RoboDK station: Entorno1_4clases.rdk

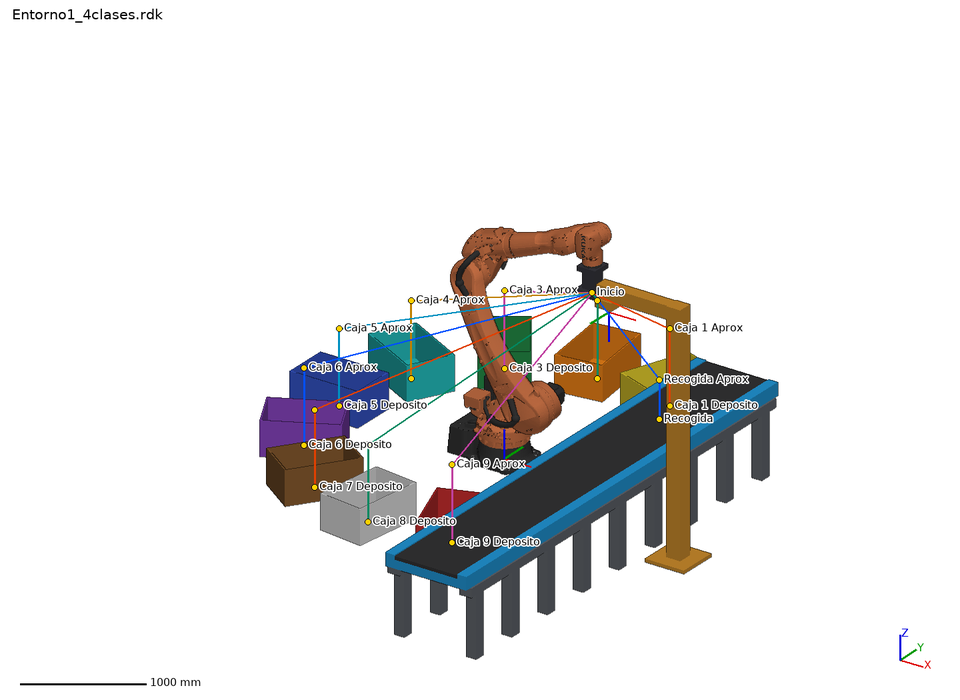
[picture v0: the station drawn from its stored meshes, robots at their saved joint values, targets as dots, program paths as lines]
Station Entorno1 (saved by RoboDK 5.9.0). Poses are relative to the parent item; angles as X-Y-Z fixed-axis rotations.
Station parameters (name, value as stored): BandaEstado, OFF, PRUEBA_LLAMADA, fin, TIPO_B0, 0, TIPO_B1, 1, TIPO_B2, 0, TIPO_B3, 0, TIPO_VALIDO, 0, HOJA_EN_CAMARA, 0, ORDEN_RECIBIDA, 0, ROBOT_OCUPADO, 0, CAJA_DESTINO, 2, ULTIMO_CODIGO, 2, VENTOSA, 0, CONTROL, RUN, IMAGEN_HOJA, C:/Users/edgar/OneDrive/Escritorio/RoboDK\camara_hoja_actual.png, HOJA_ID, 20260911_153832767_iOS
  - frame KUKA IONTEC ultra KR 120 R2700 Base at (0, 0, 0) mm
    - robot KUKA IONTEC ultra KR 120 R2700: 6 axes
        modified DH rows (alpha deg, a mm, theta deg, d mm): 0, 0, 0, 575; -90, 330, 0, 0; 0, 1180, -90, 0; -90, 170, 0, 1180; 90, 0, 0, 0; -90, 0, 180, 230
        joint limits [-185, -140, -95, -180, -125, -350] to [185, 60, 171, 180, 125, 350]; home [0, -90, 90, 0, 0, 0]; saved at [0, -117, 97.5, 0, 109.5, 0]
      - tool Ventosa, TCP at (0, 0, 250) mm, size 200 x 200 x 250 mm
  - object Banda at (0, 0, 0) mm, size 606 x 4306 x 30 mm
  - object Banda Bastidor at (0, 0, 0) mm, size 786 x 4306 x 120 mm
  - object Soporte Banda at (0, 0, 0) mm, size 816 x 4206 x 656.5 mm
  - object Estructura Camara at (0, 0, 0) mm, size 940 x 380 x 2242.1 mm
    - frame Camara Ref at (1500, -700, 1992.06) mm, rotated rx 180 ry 0 rz 0 deg
  - camera Camara Banda
  - object Caja 1 at (547.23, 1503.51, 0) mm, rotated rx 0 ry 0 rz 70 deg, size 660 x 430 x 320 mm
  - object Caja 2 at (-208.84, 1586.31, 0) mm, rotated rx 0 ry 0 rz 97.5 deg, size 660 x 430 x 320 mm
    - object Hoja 5 - connecticut capa at (-277.68, 0, 15) mm, rotated rx 0 ry 0 rz -90 deg, size 264.4 x 555.4 x 0.3 mm, geometry from 20260911_152855641_iOS.obj
    - object Hoja 6 - connecticut capa at (-259.95, 0, 15) mm, rotated rx 0 ry 0 rz -90 deg, size 208.9 x 519.9 x 0.3 mm, geometry from 20260911_153551286_iOS.obj
    - object Hoja 10 - connecticut capa at (-280.67, 0, 15) mm, rotated rx 0 ry 0 rz -90 deg, size 309.3 x 561.3 x 0.3 mm, geometry from 20260911_152611302_iOS.obj
    - object Hoja 14 - connecticut capa at (-290.65, 0, 15) mm, rotated rx 0 ry 0 rz -90 deg, size 317.9 x 581.3 x 0.3 mm, geometry from 20260911_152947681_iOS.obj
    - object Hoja 15 - connecticut capa at (-210.73, 0, 15) mm, rotated rx 0 ry 0 rz -90 deg, size 202 x 421.5 x 0.3 mm, geometry from 20260911_152212891_iOS.obj
    - object Hoja 16 - connecticut capa at (-248.11, 0, 15) mm, rotated rx 0 ry 0 rz -90 deg, size 209.5 x 496.2 x 0.3 mm, geometry from 20260911_154449975_iOS.obj
    - object Hoja 17 - connecticut capa at (-297.04, 0, 15) mm, rotated rx 0 ry 0 rz -90 deg, size 321 x 594.1 x 0.3 mm, geometry from 20260911_152508518_iOS.obj
    - object Hoja 18 - connecticut capa at (-263.19, 0, 15) mm, rotated rx 0 ry 0 rz -90 deg, size 219.7 x 526.4 x 0.3 mm, geometry from 20260911_152643389_iOS.obj
    - object Hoja 20 - connecticut capa at (-262.17, 0, 15) mm, rotated rx 0 ry 0 rz -90 deg, size 238.9 x 524.3 x 0.3 mm, geometry from 20260911_153832767_iOS.obj
  - object Caja 3 at (-917.72, 1310.64, 0) mm, rotated rx 0 ry 0 rz 125 deg, size 660 x 430 x 320 mm
    - object Hoja 1 - connecticut xl_izq at (-252.38, 0, 15) mm, rotated rx 0 ry 0 rz -90 deg, size 223.1 x 504.8 x 0.3 mm, geometry from 20260911_160812762_iOS.obj
    - object Hoja 7 - connecticut xl_izq at (-285.08, 0, 15) mm, rotated rx 0 ry 0 rz -90 deg, size 179.8 x 570.2 x 0.3 mm, geometry from 20260911_160352812_iOS.obj
    - object Hoja 13 - connecticut xl_izq at (-242.13, 0, 15) mm, rotated rx 0 ry 0 rz -90 deg, size 175.8 x 484.3 x 0.3 mm, geometry from 20260911_155539515_iOS.obj
  - object Caja 4 at (-1419.22, 738.8, 0) mm, rotated rx 0 ry 0 rz 152.5 deg, size 660 x 430 x 320 mm
    - object Hoja 9 - connecticut xr_der at (-263.12, 0, 15) mm, rotated rx 0 ry 0 rz -90 deg, size 209.2 x 526.2 x 0.3 mm, geometry from 20260911_161335259_iOS.obj
  - object Caja 5 at (-1600, 0, 0) mm, rotated rx 0 ry 0 rz 180 deg, size 660 x 430 x 320 mm
  - object Caja 6 at (-1419.22, -738.8, 0) mm, rotated rx 0 ry 0 rz -152.5 deg, size 660 x 430 x 320 mm
  - object Caja 7 at (-917.72, -1310.64, 0) mm, rotated rx 0 ry 0 rz -125 deg, size 660 x 430 x 320 mm
  - object Caja 8 at (-208.84, -1586.31, 0) mm, rotated rx 0 ry 0 rz -97.5 deg, size 660 x 430 x 320 mm
  - object Caja 9 at (547.23, -1503.51, 0) mm, rotated rx 0 ry 0 rz -70 deg, size 660 x 430 x 320 mm
    - object Hoja 2 - connecticut xl_izq at (-271.25, 0, 15) mm, rotated rx 0 ry 0 rz -90 deg, size 221.9 x 542.5 x 0.3 mm, geometry from 20260911_160413627_iOS.obj
    - object Hoja 3 - connecticut xr_der at (-283.84, 0, 15) mm, rotated rx 0 ry 0 rz -90 deg, size 206.1 x 567.7 x 0.3 mm, geometry from 20260911_161114446_iOS.obj
    - object Hoja 4 - connecticut xr_der at (-251.64, 0, 15) mm, rotated rx 0 ry 0 rz -90 deg, size 209.9 x 503.3 x 0.3 mm, geometry from 20260911_161042953_iOS.obj
    - object Hoja 8 - connecticut xl_izq at (-249.2, 0, 15) mm, rotated rx 0 ry 0 rz -90 deg, size 190.4 x 498.4 x 0.3 mm, geometry from 20260911_160151563_iOS.obj
    - object Hoja 11 - connecticut xr_der at (-278.06, 0, 15) mm, rotated rx 0 ry 0 rz -90 deg, size 229.2 x 556.1 x 0.3 mm, geometry from 20260911_161421883_iOS.obj
    - object Hoja 12 - connecticut capa at (-311.99, 0, 15) mm, rotated rx 0 ry 0 rz -90 deg, size 292.7 x 624 x 0.3 mm, geometry from 20260911_153901232_iOS.obj
    - object Hoja 19 - connecticut capa at (-288.58, 0, 15) mm, rotated rx 0 ry 0 rz -90 deg, size 283.4 x 577.2 x 0.3 mm, geometry from 20260911_152749963_iOS.obj
  - frame Marco Celda at (0, 0, 0) mm
    - target Inicio (joint target) at (849.86, 0, 1700.53) mm, rotated rx 180 ry 0 rz -180 deg; joints [0, -117, 97.5, 0, 109.5, 0] of KUKA IONTEC ultra KR 120 R2700
    - target Recogida Aprox (Cartesian target) at (1500, 0, 1116.8) mm, rotated rx 180 ry 0 rz 0 deg; joints [0, -90.566, 106.386, 0, 74.179, -180] of KUKA IONTEC ultra KR 120 R2700
    - target Recogida (Cartesian target) at (1500, 0, 766.8) mm, rotated rx 180 ry 0 rz 0 deg; joints [0, -85.628, 118.876, 0, 56.753, -180] of KUKA IONTEC ultra KR 120 R2700
    - target Caja 1 Aprox (Cartesian target) at (547.23, 1503.51, 700) mm, rotated rx 180 ry 0 rz -20 deg; joints [-70, -79.501, 115.457, 0, 54.044, 90] of KUKA IONTEC ultra KR 120 R2700
    - target Caja 1 Deposito (Cartesian target) at (547.23, 1503.51, 15.3) mm, rotated rx 180 ry 0 rz -20 deg; joints [-70, -54.433, 123.319, 0, 21.113, 90] of KUKA IONTEC ultra KR 120 R2700
    - target Caja 2 Aprox (Cartesian target) at (-208.84, 1586.31, 700) mm, rotated rx 180 ry 0 rz 7.5 deg; joints [-97.5, -79.501, 115.457, 0, 54.044, 90] of KUKA IONTEC ultra KR 120 R2700
    - target Caja 2 Deposito (Cartesian target) at (-208.84, 1586.31, 15.3) mm, rotated rx 180 ry 0 rz 7.5 deg; joints [-97.5, -54.433, 123.319, 0, 21.113, 90] of KUKA IONTEC ultra KR 120 R2700
    - target Caja 3 Aprox (Cartesian target) at (-917.72, 1310.64, 700) mm, rotated rx 180 ry 0 rz 35 deg; joints [-125, -79.501, 115.457, 0, 54.044, 90] of KUKA IONTEC ultra KR 120 R2700
    - target Caja 3 Deposito (Cartesian target) at (-917.72, 1310.64, 15.3) mm, rotated rx 180 ry 0 rz 35 deg; joints [-125, -54.433, 123.319, 0, 21.113, 90] of KUKA IONTEC ultra KR 120 R2700
    - target Caja 4 Aprox (Cartesian target) at (-1419.22, 738.8, 700) mm, rotated rx 180 ry 0 rz 62.5 deg; joints [-152.5, -79.501, 115.457, 0, 54.044, 90] of KUKA IONTEC ultra KR 120 R2700
    - target Caja 4 Deposito (Cartesian target) at (-1419.22, 738.8, 15.3) mm, rotated rx 180 ry 0 rz 62.5 deg; joints [-152.5, -54.433, 123.319, 0, 21.113, 90] of KUKA IONTEC ultra KR 120 R2700
    - target Caja 5 Aprox (Cartesian target) at (-1600, 0, 700) mm, rotated rx 180 ry 0 rz 90 deg; joints [-180, -79.501, 115.457, 0, 54.044, 90] of KUKA IONTEC ultra KR 120 R2700
    - target Caja 5 Deposito (Cartesian target) at (-1600, 0, 15.3) mm, rotated rx 180 ry 0 rz 90 deg; joints [-180, -54.433, 123.319, 0, 21.113, 90] of KUKA IONTEC ultra KR 120 R2700
    - target Caja 6 Aprox (Cartesian target) at (-1419.22, -738.8, 700) mm, rotated rx 180 ry 0 rz 117.5 deg; joints [152.5, -79.501, 115.457, 0, 54.044, 90] of KUKA IONTEC ultra KR 120 R2700
    - target Caja 6 Deposito (Cartesian target) at (-1419.22, -738.8, 15.3) mm, rotated rx 180 ry 0 rz 117.5 deg; joints [152.5, -54.433, 123.319, 0, 21.113, 90] of KUKA IONTEC ultra KR 120 R2700
    - target Caja 7 Aprox (Cartesian target) at (-917.72, -1310.64, 700) mm, rotated rx 180 ry 0 rz 145 deg; joints [125, -79.501, 115.457, 0, 54.044, 90] of KUKA IONTEC ultra KR 120 R2700
    - target Caja 7 Deposito (Cartesian target) at (-917.72, -1310.64, 15.3) mm, rotated rx 180 ry 0 rz 145 deg; joints [125, -54.433, 123.319, 0, 21.113, 90] of KUKA IONTEC ultra KR 120 R2700
    - target Caja 8 Aprox (Cartesian target) at (-208.84, -1586.31, 700) mm, rotated rx 180 ry 0 rz 172.5 deg; joints [97.5, -79.501, 115.457, 0, 54.044, 90] of KUKA IONTEC ultra KR 120 R2700
    - target Caja 8 Deposito (Cartesian target) at (-208.84, -1586.31, 15.3) mm, rotated rx 180 ry 0 rz 172.5 deg; joints [97.5, -54.433, 123.319, 0, 21.113, 90] of KUKA IONTEC ultra KR 120 R2700
    - target Caja 9 Aprox (Cartesian target) at (547.23, -1503.51, 700) mm, rotated rx 180 ry 0 rz -160 deg; joints [70, -79.501, 115.457, 0, 54.044, 90] of KUKA IONTEC ultra KR 120 R2700
    - target Caja 9 Deposito (Cartesian target) at (547.23, -1503.51, 15.3) mm, rotated rx 180 ry 0 rz -160 deg; joints [70, -54.433, 123.319, 0, 21.113, 90] of KUKA IONTEC ultra KR 120 R2700
  - frame Hojas Patron at (0, 0, -3000) mm
    - object Patron connecticut banda at (0, 0, 0) mm, size 236.1 x 483 x 0.3 mm
    - object Patron connecticut capa at (0, 0, 0) mm, size 184.6 x 419.9 x 0.3 mm
    - object Patron connecticut xl_izq at (0, 0, 0) mm, size 241.9 x 529.8 x 0.3 mm
    - object Patron connecticut xr_der at (0, 0, 0) mm, size 225.5 x 438.5 x 0.3 mm
    - object Patron habano banda at (0, 0, 0) mm, size 290.2 x 553.2 x 0.3 mm
    - object Patron habano capa at (0, 0, 0) mm, size 220.5 x 538.1 x 0.3 mm
    - object Patron habano xl_izq at (0, 0, 0) mm, size 259.2 x 534.9 x 0.3 mm
    - object Patron habano xr_der at (0, 0, 0) mm, size 239.2 x 491.4 x 0.3 mm
  - Python program Control_Senales (listed below)
  - Python program Ventosa_Agarrar (listed below)
  - Python program Ventosa_Soltar (listed below)
  - Python program Banda_ON (listed below)
  - Python program Banda_OFF (listed below)
  - Python program Alimentar_Pieza (listed below)
  - Python program Ciclo_Pick_Place (listed below)
  - Python program Reset_Celda (listed below)
  - program Recoger_Hoja (9 instructions, listed below)
  - program Dejar_Caja_01 (9 instructions, listed below)
  - program Dejar_Caja_02 (9 instructions, listed below)
  - program Dejar_Caja_03 (9 instructions, listed below)
  - program Dejar_Caja_04 (9 instructions, listed below)
  - program Dejar_Caja_05 (9 instructions, listed below)
  - program Dejar_Caja_06 (9 instructions, listed below)
  - program Dejar_Caja_07 (9 instructions, listed below)
  - program Dejar_Caja_08 (9 instructions, listed below)
  - program Dejar_Caja_09 (9 instructions, listed below)
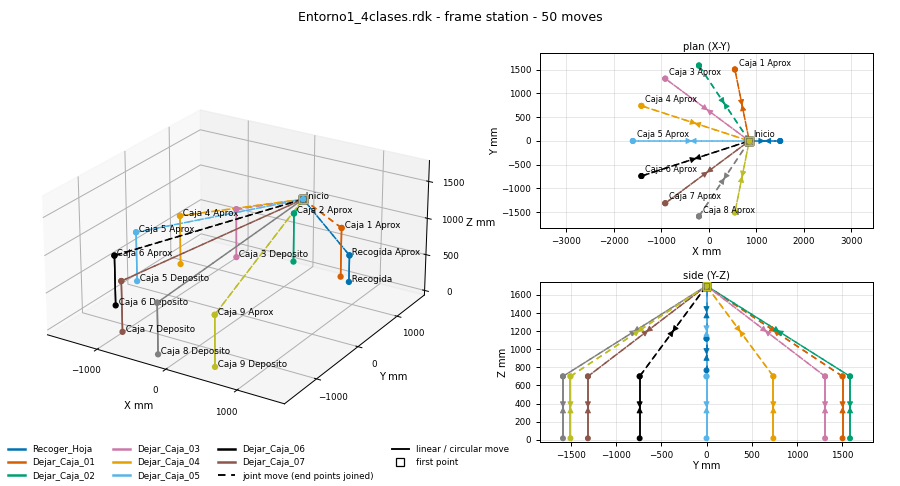
[picture p0: tool path of Entorno1_4clases.rdk in frame station, 50 of 50 moves have a stored position in this frame; points joined in program order, loops and branches not executed]

--- Python program Control_Senales ---
# Programa principal de la celda controlada por senales (modelo agentico).
#
# Ciclo por hoja:
#   1. Coloca al azar una hoja al inicio de la linea y la lleva hasta la camara.
#   2. Para la banda bajo la camara (minimo 3 s), guarda la imagen y pone
#      HOJA_EN_CAMARA = 1: el agente ya puede clasificarla.
#   3. Espera la orden del agente: codigo de 4 bits (TIPO_B0..TIPO_B3) + TIPO_VALIDO.
#   4. Acusa recibo (ORDEN_RECIBIDA = 1), lleva la hoja a la zona de recogida y
#      ejecuta los programas de robot Recoger_Hoja y Dejar_Caja_NN.
#   5. Anota el resultado en registro_clasificacion.csv.
#
# Codigos:  1..8 -> caja del tipo de hoja   |   9 -> caja 9 (no reconocida)
#           0 y 10..15 (no validos) -> caja 9, para no perder la hoja.
#
# Para detenerlo de forma ordenada: poner el parametro CONTROL = STOP. Solo se atiende en
# puntos seguros (esperando orden o entre ciclos): si llega con el robot en movimiento,
# se termina la hoja en curso, se anota y despues se para.
import os
import random
import time
from robodk.robolink import *
from robodk.robomath import *

RDK = Robolink()

robot = RDK.Item('KUKA IONTEC ultra KR 120 R2700', ITEM_TYPE_ROBOT)
tool = RDK.Item('Ventosa', ITEM_TYPE_TOOL)
marco = RDK.Item('Marco Celda', ITEM_TYPE_FRAME)
banda = RDK.Item('Banda', ITEM_TYPE_OBJECT)
camref = RDK.Item('Camara Ref', ITEM_TYPE_FRAME)
camara = RDK.Item('Camara Banda', ITEM_TYPE_CAMERA)

# --- geometria de la linea (igual que en Construir_Entorno.py)
BELT_CX = 1500.0
BELT_TOP = 766.5
BELT_Y0 = -3229.5            # inicio de la linea
CAM_Y = -700.0               # camara
Y_RECOGIDA = 0.0             # zona de recogida
VEL_BANDA = 300.0            # mm/s
REFRESCO = 0.02
PARADA_MIN_CAMARA = 3.0      # s minimos bajo la camara (tiempo de simulacion)
CAM_PARAMS = 'FOCAL_LENGTH=6 FOV=28.39 FAR_LENGTH=2500 SIZE=640x480'

# --- tipos de hoja: tipo N -> caja N. Mismo orden que CLASES en Construir_Entorno.py
CLASES = ['connecticut banda', 'connecticut capa',
          'connecticut xl_izq', 'connecticut xr_der',
          'habano banda', 'habano capa',
          'habano xl_izq', 'habano xr_der']
CAJA_ESPECIAL = 9
N_HOJAS = 0                  # 0 = sin fin (o hasta agotar la cola, si la hay)

# La carpeta se averigua, no se clava: la ruta escrita era la de otra maquina
# (C:\Users\LENOVO\Desktop\RoboDK) y aqui el usuario es otro, asi que la imagen de
# la camara y el registro se escribian en un sitio que no existe -- y
# `guardar_imagen` se lo tragaba en silencio por su try/except.
def _carpeta():
    try:
        est = str(RDK.getParam('PATH_OPENSTATION'))
        if os.path.isdir(est):
            return est
    except Exception:
        pass
    try:
        return os.path.dirname(os.path.dirname(os.path.abspath(__file__)))
    except Exception:
        return os.path.expanduser('~')


CARPETA = _carpeta()
IMAGEN = os.path.join(CARPETA, 'camara_hoja_actual.png')
REGISTRO = os.path.join(CARPETA, 'registro_clasificacion.csv')

# La cola de hojas que prepara el agente (`scripts/cola_entorno1.py`). Si existe,
# las hojas salen EN ESE ORDEN y con su malla propia; si no, se alimenta al azar
# con las diez hojas patron, que es como estaba.
COLA = r'D:\tesis-tabaco\out\celda\entorno1\cola_hojas.csv'

ENTRADAS = ['TIPO_B0', 'TIPO_B1', 'TIPO_B2', 'TIPO_B3', 'TIPO_VALIDO']
SALIDAS = ['HOJA_EN_CAMARA', 'ORDEN_RECIBIDA', 'ROBOT_OCUPADO', 'CAJA_DESTINO', 'ULTIMO_CODIGO']


class Detenido(Exception):
    pass


def leer_cola():
    '''Las hojas a pasar, en orden. Lista vacia = alimentar al azar, como antes.'''
    if not os.path.isfile(COLA):
        return []
    import csv
    with open(COLA, encoding='utf-8') as f:
        return [r for r in csv.DictReader(f, delimiter=';') if r.get('obj')]


COLA_FILAS = leer_cola()
COLA_I = [0]                 # en lista para poder tocarlo desde alimentar()


# ----------------------------------------------------------------- senales
def leer(nombre):
    try:
        return int(float(str(RDK.getParam(nombre)).strip()))
    except (TypeError, ValueError):
        return 0


def escribir(nombre, valor):
    RDK.setParam(nombre, str(int(valor)))


def parada_pedida():
    return str(RDK.getParam('CONTROL')).strip().upper() == 'STOP'


def comprobar_parada():
    """Solo se llama en puntos seguros (sin hoja en la ventosa ni robot en movimiento)."""
    if parada_pedida():
        raise Detenido()


def leer_codigo():
    """Compone el codigo de 4 bits: B0 es el bit menos significativo."""
    return sum((leer('TIPO_B%i' % k) & 1) << k for k in range(4))


def codigo_a_caja(codigo):
    if 1 <= codigo <= len(CLASES):
        return codigo
    return CAJA_ESPECIAL          # 9 = no reconocida; 0 y 10..15 = no validos


def cerrar_handshake():
    """Fase 4: cuando el agente baja TIPO_VALIDO, el robot baja ORDEN_RECIBIDA."""
    if leer('ORDEN_RECIBIDA') == 1 and leer('TIPO_VALIDO') == 0:
        escribir('ORDEN_RECIBIDA', 0)


# ----------------------------------------------------------------- tiempo
def esperar_sim(segundos):
    """Espera en tiempo de simulacion (escala con la velocidad de simulacion)."""
    tic()
    t_ant, t = toc(), 0.0
    while t < segundos:
        comprobar_parada()
        t_act = toc()
        t += (t_act - t_ant) * RDK.SimulationSpeed()
        t_ant = t_act
        pause(REFRESCO)


# ----------------------------------------------------------------- hojas y banda
def centro_y(obj):
    """El origen de la hoja esta en su lado corto: el centro sale del bounding box."""
    bb = obj.setParam('BoundingBox')
    return (bb['min'][1] + bb['max'][1]) / 2.0


def siguiente_numero():
    usados = []
    for o in RDK.ItemList(ITEM_TYPE_OBJECT):
        if o.Name().startswith('Hoja '):
            try:
                usados.append(int(o.Name().split()[1]))
            except ValueError:
                pass
    return max(usados) + 1 if usados else 1


def coloca(hoja, clase, ident):
    '''Nombra la hoja y publica su identificador para el agente.

    `HOJA_ID` es el nombre del fichero de su FOTO, que no dice la clase: es lo
    que el agente usa para encontrar la fotografia real. El nombre del objeto si
    lleva la etiqueta, y el agente NO lo lee -- leerla es lo que hacia que la
    celda "clasificara" sin clasificar.
    '''
    hoja.setName('Hoja %i - %s' % (siguiente_numero(), clase))
    RDK.setParam('HOJA_ID', ident)


def alimentar():
    '''Saca la siguiente hoja de la cola; si no hay cola, una patron al azar.'''
    if COLA_FILAS and COLA_I[0] < len(COLA_FILAS):
        r = COLA_FILAS[COLA_I[0]]
        COLA_I[0] += 1
        clase = '%s %s' % (r['variedad'], r['clase'])
        tipo_real = CLASES.index(clase) + 1 if clase in CLASES else 0
        hoja = RDK.AddFile(r['obj'], marco)
        if not hoja.Valid():
            raise Exception('RoboDK no pudo cargar la malla: ' + r['obj'])
        coloca(hoja, clase, r['id'])
        hoja.setPoseAbs(transl(BELT_CX, BELT_Y0, BELT_TOP))
        hoja.setVisible(True)
        RDK.setCollisionActivePair(COLLISION_OFF, tool, hoja)
        RDK.setCollisionActivePair(COLLISION_OFF, banda, hoja)
        for c in RDK.ItemList(ITEM_TYPE_OBJECT):
            if c.Name().startswith('Caja '):
                RDK.setCollisionActivePair(COLLISION_OFF, c, hoja)
        return hoja, clase, tipo_real

    tipo_real = random.randint(1, len(CLASES))
    clase = CLASES[tipo_real - 1]
    patron = RDK.Item('Patron ' + clase, ITEM_TYPE_OBJECT)
    if not patron.Valid():
        raise Exception('Falta la hoja patron: ' + clase)
    RDK.Copy(patron)
    hoja = RDK.Paste(marco)
    coloca(hoja, clase, '')
    hoja.setPoseAbs(transl(BELT_CX, BELT_Y0, BELT_TOP))
    hoja.setVisible(True)
    # Contactos previstos por diseno: no deben marcarse como colision.
    RDK.setCollisionActivePair(COLLISION_OFF, tool, hoja)
    RDK.setCollisionActivePair(COLLISION_OFF, banda, hoja)
    for c in RDK.ItemList(ITEM_TYPE_OBJECT):
        if c.Name().startswith('Caja '):
            RDK.setCollisionActivePair(COLLISION_OFF, c, hoja)
    return hoja, clase, tipo_real


def transportar(hoja, y_destino):
    """Banda en marcha hasta que el CENTRO de la hoja llega a y_destino.
    No se interrumpe: una parada pedida se atiende al llegar."""
    RDK.setParam('BandaEstado', 'ON')
    tic()
    t_ant = toc()
    while True:
        cerrar_handshake()
        t_act = toc()
        dt = (t_act - t_ant) * RDK.SimulationSpeed()
        t_ant = t_act
        x, y, z = hoja.PoseAbs().Pos()
        falta = y_destino - centro_y(hoja)
        if falta <= VEL_BANDA * dt:
            hoja.setPoseAbs(transl(x, y + falta, z))
            break
        hoja.setPoseAbs(transl(x, y + VEL_BANDA * dt, z))
        pause(REFRESCO)
    RDK.setParam('BandaEstado', 'OFF')


def guardar_imagen(cam):
    """Deja la imagen de la camara en disco para quien la necesite."""
    try:
        if RDK.Cam2D_Snapshot(IMAGEN, cam):
            RDK.setParam('IMAGEN_HOJA', IMAGEN)
    except Exception:
        pass


# ----------------------------------------------------------------- robot
def ejecutar(nombre):
    """Lanza un programa de robot y espera a que termine. No se interrumpe."""
    prog = RDK.Item(nombre, ITEM_TYPE_PROGRAM)
    if not prog.Valid():
        raise Exception('No existe el programa de robot: ' + nombre)
    prog.RunProgram()
    t0 = time.time()
    while not prog.Busy() and time.time() - t0 < 2.0:
        pause(0.02)
    while prog.Busy():
        cerrar_handshake()
        pause(0.05)


def esperar_orden():
    """Pide clasificacion y espera el codigo de 4 bits del agente."""
    # El handshake anterior tiene que estar cerrado antes de pedir otra orden.
    while leer('TIPO_VALIDO') == 1:
        comprobar_parada()
        pause(0.05)
    escribir('ORDEN_RECIBIDA', 0)

    escribir('HOJA_EN_CAMARA', 1)
    RDK.Command('SilentMessage', 'Hoja bajo la camara: esperando el tipo (4 bits)')
    esperar_sim(PARADA_MIN_CAMARA)          # inspeccion minima de 3 s
    while leer('TIPO_VALIDO') != 1:
        comprobar_parada()
        pause(0.05)
    codigo = leer_codigo()
    escribir('ORDEN_RECIBIDA', 1)
    escribir('HOJA_EN_CAMARA', 0)
    return codigo


def registrar(hoja, clase, tipo_real, codigo, caja):
    nuevo = not os.path.isfile(REGISTRO)
    if tipo_real == 0:
        # Hoja sin etiqueta: no hay verdad de campo contra la que puntuar, y
        # decir ACIERTO o ERROR seria inventarsela.
        resultado = 'SIN_ETIQUETA'
    elif codigo == tipo_real:
        resultado = 'ACIERTO'
    elif caja == CAJA_ESPECIAL:
        resultado = 'ESPECIAL'
    else:
        resultado = 'ERROR'
    with open(REGISTRO, 'a', encoding='utf-8') as f:
        if nuevo:
            f.write('fecha;hoja;clase_real;tipo_real;codigo_recibido;bits_B3_B0;caja;resultado\n')
        f.write('%s;%s;%s;%i;%i;%s;%i;%s\n' % (
            time.strftime('%Y-%m-%d %H:%M:%S'), hoja.Name(), clase, tipo_real,
            codigo, format(codigo, '04b'), caja, resultado))
    return resultado


# ----------------------------------------------------------------- programa principal
for n in ENTRADAS + SALIDAS:
    escribir(n, 0)
RDK.setParam('CONTROL', 'RUN')

robot.setPoseFrame(marco)
robot.setPoseTool(tool)
robot.MoveJ(RDK.Item('Inicio', ITEM_TYPE_TARGET))

# La imagen solo sale bien si la vista se abre desde este mismo proceso.
cam = camara
try:
    RDK.Cam2D_Close()
    cam = RDK.Cam2D_Add(camref, CAM_PARAMS, camara)
    cam.setName('Camara Banda')
except Exception:
    pass

n = 0
try:
    cola_agotada = lambda: bool(COLA_FILAS) and COLA_I[0] >= len(COLA_FILAS)
    while (N_HOJAS == 0 or n < N_HOJAS) and not cola_agotada():
        comprobar_parada()                      # punto seguro: entre hojas
        n += 1
        hoja, clase, tipo_real = alimentar()
        transportar(hoja, CAM_Y)
        guardar_imagen(cam)

        codigo = esperar_orden()                # punto seguro: esperando al agente
        caja = codigo_a_caja(codigo)
        escribir('ULTIMO_CODIGO', codigo)
        escribir('CAJA_DESTINO', caja)
        escribir('ROBOT_OCUPADO', 1)
        RDK.Command('SilentMessage', 'Orden %s (codigo %i) -> Caja %i' % (format(codigo, '04b'), codigo, caja))

        # Desde aqui la hoja se termina siempre, aunque se pida parar.
        transportar(hoja, Y_RECOGIDA)
        ejecutar('Recoger_Hoja')
        ejecutar('Dejar_Caja_%02d' % caja)

        escribir('ROBOT_OCUPADO', 0)
        resultado = registrar(hoja, clase, tipo_real, codigo, caja)
        RDK.Command('SilentMessage', '%s: %s -> Caja %i (%s)' % (hoja.Name(), clase, caja, resultado))
except Detenido:
    RDK.Command('SilentMessage', 'Control_Senales detenido')
finally:
    RDK.setParam('BandaEstado', 'OFF')
    escribir('HOJA_EN_CAMARA', 0)
    escribir('ROBOT_OCUPADO', 0)

--- Python program Ventosa_Agarrar ---
# Macro de la ventosa: AGARRAR.
# La llaman los programas de robot (Recoger_Hoja) justo cuando el TCP toca la hoja.
# En el robot real equivale a activar la salida de vacio.
from robodk.robolink import *
from robodk.robomath import *

RDK = Robolink()
robot = RDK.Item('KUKA IONTEC ultra KR 120 R2700', ITEM_TYPE_ROBOT)
tool = RDK.Item('Ventosa', ITEM_TYPE_TOOL)

DIST_XY = 150.0      # la hoja debe estar como mucho a esta distancia del TCP en planta
DIST_Z = 20.0        # y a esta distancia en altura


def tcp_abs():
    """Posicion absoluta del TCP de la ventosa."""
    return robot.Parent().PoseAbs() * robot.SolveFK(robot.Joints(), tool.PoseTool())


def centro(obj):
    bb = obj.setParam('BoundingBox')
    return [(bb['min'][k] + bb['max'][k]) / 2.0 for k in range(3)]


tx, ty, tz = tcp_abs().Pos()
mejor, d_mejor = None, 1e9
for o in RDK.ItemList(ITEM_TYPE_OBJECT):
    if not o.Name().startswith('Hoja '):
        continue
    if o.Parent().Type() == ITEM_TYPE_TOOL or o.Parent().Name().startswith('Caja '):
        continue                              # ya agarrada o ya depositada
    cx, cy, cz = centro(o)
    dxy = ((cx - tx) ** 2 + (cy - ty) ** 2) ** 0.5
    if dxy < DIST_XY and abs(cz - tz) < DIST_Z and dxy < d_mejor:
        mejor, d_mejor = o, dxy

if mejor is None:
    RDK.setParam('VENTOSA', '0')
    RDK.Command('SilentMessage', 'Ventosa: no hay hoja bajo la ventosa')
else:
    pose = mejor.PoseAbs()
    mejor.setParentStatic(tool)
    mejor.setPoseAbs(pose)
    RDK.setParam('VENTOSA', '1')
    RDK.Command('SilentMessage', 'Ventosa: agarrada %s' % mejor.Name())

--- Python program Ventosa_Soltar ---
# Macro de la ventosa: SOLTAR.
# La llaman los programas de robot (Dejar_Caja_NN) cuando el TCP esta dentro de la caja.
# En el robot real equivale a cortar el vacio (y soplar).
from robodk.robolink import *
from robodk.robomath import *

RDK = Robolink()
robot = RDK.Item('KUKA IONTEC ultra KR 120 R2700', ITEM_TYPE_ROBOT)
tool = RDK.Item('Ventosa', ITEM_TYPE_TOOL)
marco = RDK.Item('Marco Celda', ITEM_TYPE_FRAME)

tx, ty, tz = (robot.Parent().PoseAbs() * robot.SolveFK(robot.Joints(), tool.PoseTool())).Pos()

# Caja cuyo centro queda mas cerca del TCP en planta: ahi se queda la hoja.
caja, d_caja = None, 1e9
for o in RDK.ItemList(ITEM_TYPE_OBJECT):
    if o.Name().startswith('Caja '):
        cx, cy, _ = o.PoseAbs().Pos()
        d = ((cx - tx) ** 2 + (cy - ty) ** 2) ** 0.5
        if d < d_caja:
            caja, d_caja = o, d
destino = caja if (caja is not None and d_caja < 400.0) else marco

soltadas = []
for o in RDK.ItemList(ITEM_TYPE_OBJECT):
    if o.Name().startswith('Hoja ') and o.Parent().Type() == ITEM_TYPE_TOOL:
        pose = o.PoseAbs()
        o.setParentStatic(destino)
        o.setPoseAbs(pose)
        soltadas.append(o.Name())

RDK.setParam('VENTOSA', '0')
RDK.Command('SilentMessage', 'Ventosa: soltada(s) %s en %s' % (soltadas, destino.Name()))

--- Python program Banda_ON ---
# Enciende la banda transportadora.
#
# Mientras esta encendida arrastra hacia +Y todas las hojas que haya sobre la cinta.
# Cada hoja se detiene 3 segundos al llegar a la camara y despues sigue su camino.
# Las que llegan al final del recorrido se retiran. Se para ejecutando Banda_OFF.
# Sigue el patron de Library/Macros/RunConveyor.py de RoboDK.
from robodk.robolink import *
from robodk.robomath import *

RDK = Robolink()

BELT_CX = 1500.0
BELT_TOP = 766.5
BELT_Y0 = -3229.5             # inicio de la linea
BELT_Y1 = 1076.5              # final de la linea
CAM_Y = -700.0                # posicion de la camara
PARADA_CAMARA = 3.0           # s de parada bajo la camara (tiempo de simulacion)
VEL_BANDA = 300.0             # mm/s
REFRESCO = 0.02
ANCHO_NEGRO = 606.0


def centro_y(obj):
    """La hoja tiene el origen en su lado corto: el centro sale del bounding box."""
    bb = obj.setParam('BoundingBox')
    return (bb['min'][1] + bb['max'][1]) / 2.0


def sobre_la_cinta(obj):
    """Cuenta si la hoja esta suelta sobre la cinta (no agarrada ni ya en una caja)."""
    if obj.Parent().Type() == ITEM_TYPE_TOOL:
        return False
    x, y, z = obj.PoseAbs().Pos()
    return (abs(x - BELT_CX) < ANCHO_NEGRO / 2.0
            and BELT_Y0 - 200.0 < y < BELT_Y1
            and abs(z - BELT_TOP) < 50.0)


RDK.setParam('BandaEstado', 'ON')
RDK.Command('SilentMessage', 'Banda ENCENDIDA')

inspeccionadas = set()        # hojas que ya hicieron su parada bajo la camara
espera_hasta = 0.0            # tiempo de simulacion hasta el que la banda esta parada
t_sim = 0.0

tic()
t_ant = toc()
while str(RDK.getParam('BandaEstado')).find('ON') >= 0:
    t_act = toc()
    dt = (t_act - t_ant) * RDK.SimulationSpeed()
    t_ant = t_act
    t_sim += dt

    hojas = [o for o in RDK.ItemList(ITEM_TYPE_OBJECT)
             if o.Name().startswith('Hoja ') and sobre_la_cinta(o)]

    # Parada bajo la camara: la primera hoja que llega detiene la linea 3 s
    if t_sim < espera_hasta:
        pause(REFRESCO)
        continue
    for h in hojas:
        if h.Name() not in inspeccionadas and centro_y(h) >= CAM_Y:
            inspeccionadas.add(h.Name())
            espera_hasta = t_sim + PARADA_CAMARA
            RDK.Command('SilentMessage', 'Inspeccionando %s (3 s)' % h.Name())
            break
    if t_sim < espera_hasta:
        continue

    items, poses = [], []
    for h in hojas:
        x, y, z = h.PoseAbs().Pos()
        y_nueva = y + VEL_BANDA * dt
        if centro_y(h) + VEL_BANDA * dt > BELT_Y1:
            h.Delete()                 # la hoja sale de la linea
            continue
        items.append(h)
        poses.append(transl(x, y_nueva, z))

    if items:
        RDK.setPosesAbs(items, poses)
    pause(REFRESCO)

RDK.Command('SilentMessage', 'Banda APAGADA')

--- Python program Banda_OFF ---
# Apaga la banda transportadora: las piezas se quedan donde esten.
# El bucle de Banda_ON lee esta variable y termina solo.
from robodk.robolink import *

RDK = Robolink()
RDK.setParam('BandaEstado', 'OFF')
RDK.Command('SilentMessage', 'Banda APAGADA')

--- Python program Alimentar_Pieza ---
# Coloca una hoja NUEVA AL AZAR al inicio de la linea de transporte.
# Con la banda encendida (Banda_ON) la hoja recorre la linea, se detiene 3 s bajo la
# camara y sigue hasta la zona de recogida.
import random
from robodk.robolink import *
from robodk.robomath import *

RDK = Robolink()

BELT_CX = 1500.0
BELT_TOP = 766.5
BELT_Y0 = -3229.5             # inicio de la linea

marco = RDK.Item('Marco Celda', ITEM_TYPE_FRAME)

patrones = [o for o in RDK.ItemList(ITEM_TYPE_OBJECT) if o.Name().startswith('Patron ')]
if not patrones:
    raise Exception('No hay hojas patron en la estacion. Ejecuta Construir_Entorno.py')

elegido = random.choice(patrones)
clase = elegido.Name()[len('Patron '):]

usados = []
for o in RDK.ItemList(ITEM_TYPE_OBJECT):
    if o.Name().startswith('Hoja '):
        try:
            usados.append(int(o.Name().split()[1]))
        except ValueError:
            pass
n = max(usados) + 1 if usados else 1

RDK.Copy(elegido)
hoja = RDK.Paste(marco)
hoja.setName('Hoja %i - %s' % (n, clase))    # la clase queda a la vista en el arbol
# El origen de la hoja esta en el centro de su lado corto, no en su centro.
hoja.setPoseAbs(transl(BELT_CX, BELT_Y0, BELT_TOP))
hoja.setVisible(True)

# Contactos previstos por diseno: la hoja se apoya en la cinta y la agarra la ventosa.
RDK.setCollisionActivePair(COLLISION_OFF, RDK.Item('Banda', ITEM_TYPE_OBJECT), hoja)
RDK.setCollisionActivePair(COLLISION_OFF, RDK.Item('Ventosa', ITEM_TYPE_TOOL), hoja)
for k in range(1, 31):
    caja = RDK.Item('Caja %i' % k, ITEM_TYPE_OBJECT)
    if caja.Valid():
        RDK.setCollisionActivePair(COLLISION_OFF, caja, hoja)

RDK.Command('SilentMessage', 'Hoja %i al inicio de la linea: %s' % (n, clase))

--- Python program Ciclo_Pick_Place ---
# Ciclo completo de la celda de clasificacion de hojas:
#   1. Coloca al azar una hoja al inicio de la linea.
#   2. Enciende la banda y la transporta hasta la camara.
#   3. Para la banda 3 segundos bajo la camara (inspeccion) y toma una foto.
#   4. Reanuda hasta la zona de recogida y para la banda.
#   5. El robot recoge la hoja y la deposita en la caja de su clase.
# Se repite N_CICLOS veces. Cada clase de hoja tiene su propia caja en el arco.
import random
from robodk.robolink import *
from robodk.robomath import *

RDK = Robolink()

robot = RDK.Item('KUKA IONTEC ultra KR 120 R2700', ITEM_TYPE_ROBOT)
tool = RDK.Item('Ventosa', ITEM_TYPE_TOOL)
marco = RDK.Item('Marco Celda', ITEM_TYPE_FRAME)
banda = RDK.Item('Banda', ITEM_TYPE_OBJECT)
camara = RDK.Item('Camara Banda', ITEM_TYPE_CAMERA)

BELT_CX = 1500.0
BELT_TOP = 766.5
BELT_Y0 = -3229.5           # inicio de la linea
CAM_Y = -700.0              # posicion de la camara
Y_RECOGIDA = 0.0            # zona de recogida
PARADA_CAMARA = 3.0         # s de parada bajo la camara (tiempo de simulacion)
VEL_BANDA = 300.0           # mm/s
REFRESCO = 0.02

# Orden = caja de destino. Debe coincidir con CLASES de Construir_Entorno.py.
CLASES = ['connecticut banda', 'connecticut capa', 'connecticut media_banda',
          'connecticut xl_izq', 'connecticut xr_der',
          'habano banda', 'habano capa', 'habano media_banda',
          'habano xl_izq', 'habano xr_der']
N_CICLOS = 10

robot.setPoseFrame(marco)
robot.setPoseTool(tool)
robot.setSpeed(900, 250)

T = lambda nombre: RDK.Item(nombre, ITEM_TYPE_TARGET)


def centro_y(obj):
    """La hoja tiene el origen en su lado corto: el centro sale del bounding box."""
    bb = obj.setParam('BoundingBox')
    return (bb['min'][1] + bb['max'][1]) / 2.0


def reparentar(obj, padre):
    """Cambia el padre conservando la posicion absoluta."""
    pose = obj.PoseAbs()
    obj.setParentStatic(padre)
    obj.setPoseAbs(pose)


def alimentar(n):
    """Saca al azar una copia de una hoja patron y la deja al inicio de la linea."""
    clase = random.choice(CLASES)
    patron = RDK.Item('Patron ' + clase, ITEM_TYPE_OBJECT)
    if not patron.Valid():
        raise Exception('Falta la hoja patron: ' + clase)
    RDK.Copy(patron)
    hoja = RDK.Paste(marco)
    hoja.setName('Hoja %i - %s' % (n, clase))    # la clase queda a la vista en el arbol
    hoja.setPoseAbs(transl(BELT_CX, BELT_Y0, BELT_TOP))
    hoja.setVisible(True)
    # Contactos previstos por diseno: no deben marcarse como colision.
    RDK.setCollisionActivePair(COLLISION_OFF, tool, hoja)
    RDK.setCollisionActivePair(COLLISION_OFF, banda, hoja)
    for k in range(1, len(CLASES) + 1):
        RDK.setCollisionActivePair(COLLISION_OFF, RDK.Item('Caja %i' % k, ITEM_TYPE_OBJECT), hoja)
    return hoja, clase


def transportar(hoja, y_destino):
    """Avanza la banda hasta que el CENTRO de la hoja llega a y_destino."""
    RDK.setParam('BandaEstado', 'ON')
    tic()
    t_ant = toc()
    while True:
        t_act = toc()
        dt = (t_act - t_ant) * RDK.SimulationSpeed()
        t_ant = t_act
        x, y, z = hoja.PoseAbs().Pos()
        falta = y_destino - centro_y(hoja)
        if falta <= VEL_BANDA * dt:
            hoja.setPoseAbs(transl(x, y + falta, z))
            break
        hoja.setPoseAbs(transl(x, y + VEL_BANDA * dt, z))
        pause(REFRESCO)
    RDK.setParam('BandaEstado', 'OFF')


def esperar(segundos):
    """Espera en tiempo de simulacion (se acorta si subes la velocidad de simulacion)."""
    tic()
    t_ant = toc()
    t = 0.0
    while t < segundos:
        t_act = toc()
        t += (t_act - t_ant) * RDK.SimulationSpeed()
        t_ant = t_act
        pause(REFRESCO)


for n in range(1, N_CICLOS + 1):
    hoja, clase = alimentar(n)
    caja = CLASES.index(clase) + 1
    RDK.Command('SilentMessage', 'Ciclo %i/%i: %s -> Caja %i' % (n, N_CICLOS, clase, caja))

    # --- banda ENCENDIDA hasta la camara
    transportar(hoja, CAM_Y)

    # --- parada de 3 s bajo la camara: inspeccion
    if camara.Valid():
        camara.setParam('Open')
    esperar(PARADA_CAMARA)

    # --- reanuda hasta la zona de recogida y para
    transportar(hoja, Y_RECOGIDA)

    # --- recogida
    robot.MoveJ(T('Inicio'))
    robot.MoveJ(T('Recogida Aprox'))
    robot.MoveL(T('Recogida'))
    reparentar(hoja, tool)                   # la ventosa agarra la hoja
    robot.MoveL(T('Recogida Aprox'))

    # --- traslado en postura recogida (no interfiere con la estructura de la camara)
    robot.MoveJ(T('Inicio'))
    robot.MoveJ(T('Caja %i Aprox' % caja))
    robot.MoveL(T('Caja %i Deposito' % caja))
    reparentar(hoja, RDK.Item('Caja %i' % caja, ITEM_TYPE_OBJECT))   # se suelta en la caja
    robot.MoveL(T('Caja %i Aprox' % caja))
    robot.MoveJ(T('Inicio'))

RDK.Command('SilentMessage', 'Ciclo terminado: %i hojas clasificadas' % N_CICLOS)

--- Python program Reset_Celda ---
# Devuelve la celda al estado inicial: apaga la banda, borra las piezas
# generadas y lleva el robot al target Inicio.
from robodk.robolink import *

RDK = Robolink()
RDK.setParam('BandaEstado', 'OFF')

for it in RDK.ItemList(ITEM_TYPE_OBJECT):
    if it.Name().startswith('Hoja ') or it.Name().startswith('Pieza '):
        it.Delete()

robot = RDK.Item('KUKA IONTEC ultra KR 120 R2700', ITEM_TYPE_ROBOT)
robot.setJoints(RDK.Item('Inicio', ITEM_TYPE_TARGET).Joints())
RDK.Command('SilentMessage', 'Celda reiniciada')

--- program Recoger_Hoja (robot KUKA IONTEC ultra KR 120 R2700) ---
  Est. Ref.: Marco Celda
  Est. herr: Ventosa
  Establecer velocidad (900.0 mm/s)
  MoveJ (Inicio)
  MoveJ (Recogida Aprox)
  MoveL (Recogida)
  Llamar Ventosa_Agarrar
  MoveL (Recogida Aprox)
  MoveJ (Inicio)

--- program Dejar_Caja_01 (robot KUKA IONTEC ultra KR 120 R2700) ---
  Est. Ref.: Marco Celda
  Est. herr: Ventosa
  Establecer velocidad (900.0 mm/s)
  MoveJ (Inicio)
  MoveJ (Caja 1 Aprox)
  MoveL (Caja 1 Deposito)
  Llamar Ventosa_Soltar
  MoveL (Caja 1 Aprox)
  MoveJ (Inicio)

--- program Dejar_Caja_02 (robot KUKA IONTEC ultra KR 120 R2700) ---
  Est. Ref.: Marco Celda
  Est. herr: Ventosa
  Establecer velocidad (900.0 mm/s)
  MoveJ (Inicio)
  MoveJ (Caja 2 Aprox)
  MoveL (Caja 2 Deposito)
  Llamar Ventosa_Soltar
  MoveL (Caja 2 Aprox)
  MoveJ (Inicio)

--- program Dejar_Caja_03 (robot KUKA IONTEC ultra KR 120 R2700) ---
  Est. Ref.: Marco Celda
  Est. herr: Ventosa
  Establecer velocidad (900.0 mm/s)
  MoveJ (Inicio)
  MoveJ (Caja 3 Aprox)
  MoveL (Caja 3 Deposito)
  Llamar Ventosa_Soltar
  MoveL (Caja 3 Aprox)
  MoveJ (Inicio)

--- program Dejar_Caja_04 (robot KUKA IONTEC ultra KR 120 R2700) ---
  Est. Ref.: Marco Celda
  Est. herr: Ventosa
  Establecer velocidad (900.0 mm/s)
  MoveJ (Inicio)
  MoveJ (Caja 4 Aprox)
  MoveL (Caja 4 Deposito)
  Llamar Ventosa_Soltar
  MoveL (Caja 4 Aprox)
  MoveJ (Inicio)

--- program Dejar_Caja_05 (robot KUKA IONTEC ultra KR 120 R2700) ---
  Est. Ref.: Marco Celda
  Est. herr: Ventosa
  Establecer velocidad (900.0 mm/s)
  MoveJ (Inicio)
  MoveJ (Caja 5 Aprox)
  MoveL (Caja 5 Deposito)
  Llamar Ventosa_Soltar
  MoveL (Caja 5 Aprox)
  MoveJ (Inicio)

--- program Dejar_Caja_06 (robot KUKA IONTEC ultra KR 120 R2700) ---
  Est. Ref.: Marco Celda
  Est. herr: Ventosa
  Establecer velocidad (900.0 mm/s)
  MoveJ (Inicio)
  MoveJ (Caja 6 Aprox)
  MoveL (Caja 6 Deposito)
  Llamar Ventosa_Soltar
  MoveL (Caja 6 Aprox)
  MoveJ (Inicio)

--- program Dejar_Caja_07 (robot KUKA IONTEC ultra KR 120 R2700) ---
  Est. Ref.: Marco Celda
  Est. herr: Ventosa
  Establecer velocidad (900.0 mm/s)
  MoveJ (Inicio)
  MoveJ (Caja 7 Aprox)
  MoveL (Caja 7 Deposito)
  Llamar Ventosa_Soltar
  MoveL (Caja 7 Aprox)
  MoveJ (Inicio)

--- program Dejar_Caja_08 (robot KUKA IONTEC ultra KR 120 R2700) ---
  Est. Ref.: Marco Celda
  Est. herr: Ventosa
  Establecer velocidad (900.0 mm/s)
  MoveJ (Inicio)
  MoveJ (Caja 8 Aprox)
  MoveL (Caja 8 Deposito)
  Llamar Ventosa_Soltar
  MoveL (Caja 8 Aprox)
  MoveJ (Inicio)

--- program Dejar_Caja_09 (robot KUKA IONTEC ultra KR 120 R2700) ---
  Est. Ref.: Marco Celda
  Est. herr: Ventosa
  Establecer velocidad (900.0 mm/s)
  MoveJ (Inicio)
  MoveJ (Caja 9 Aprox)
  MoveL (Caja 9 Deposito)
  Llamar Ventosa_Soltar
  MoveL (Caja 9 Aprox)
  MoveJ (Inicio)
